FUNCTION_BLOCK FB_XPlanarModule
VAR CONSTANT
	MoverCount	 : UDINT := 2;
	TrackCount	 : UDINT := 2;
	StationCount : UDINT := 2;
END_VAR

VAR
	XPlanarSystem	: FB_Component_XPlanar;
	Movers			: ARRAY[1..MoverCount] OF FB_XPlanarMover;
	Tracks			: ARRAY[1..TrackCount] OF FB_XPlanarTrackSegment;
	Stations		: ARRAY[1..StationCount] OF FB_XPlanarStationBase;
	Station1Process : FB_SimulateProcess;  //Custom process FB that can be assigned to a station
	Station2Process : FB_RotateStation;
	InitState		: (CheckForXPlanarInit, UpdateDynamics, SetStationParameters, Initialized);
END_VAR

METHOD CyclicLogic : BOOL
VAR
	i : UDINT;
END_VAR
VAR_INST
	TaskResult	: I_PlanarTaskResult;
END_VAR
XPlanarSystem.CyclicLogic();
IF NOT XPlanarSystem.Initialized THEN
	RETURN;
END_IF

//Add any logic that needs to be called every cycle here
END_METHOD

METHOD Disable : BOOL
VAR_INST
	CommandResult	: I_PlanarTaskResult;
END_VAR
CommandResult := XPlanarSystem.Abort(); // Stop Motion and Disable All Movers
IF CommandResult.Done THEN
	Disable := TRUE;
END_IF
END_METHOD

METHOD Execute : BOOL
VAR
	i : UDINT;
END_VAR
//System is 'running' cycle thru all of the stations
FOR i := 1 TO XPlanar.StationCount DO
	ip.Stations[i].Execute();
END_FOR
END_METHOD

METHOD Initialize : BOOL
VAR_INST
	i			: UDINT;
END_VAR
CASE InitState OF
	CheckForXPlanarInit: // Init Vars
		Initialize := FALSE;
		
		//Make sure the XPlanar motion system has initialized
		IF XPlanarSystem.Initialized THEN
			InitState := UpdateDynamics;
		END_IF

	UpdateDynamics: 
		//Assign Initial Application Mover Dynamics
		FOR i := 1 TO XPlanar.MoverCount DO
			ip.Movers[i].Gap						:= 200;
			ip.Movers[i].Dynamics.Movement.Velocity := GVL.MoverVelo;
			ip.Movers[i].Dynamics.Movement.Accel	:= GVL.MoverVelo * 10;
			ip.Movers[i].Dynamics.Movement.Decel	:= GVL.MoverVelo * 10;
			ip.Movers[i].Dynamics.Movement.Jerk		:= GVL.MoverVelo * 100;
			ip.Movers[i].Dynamics.Rotation.Velocity := GVL.MoverSpinVelo;
			ip.Movers[i].Dynamics.Rotation.Accel	:= GVL.MoverSpinVelo * 10;
			ip.Movers[i].Dynamics.Rotation.Decel	:= GVL.MoverSpinVelo * 10;
			ip.Movers[i].Dynamics.Rotation.Jerk		:= GVL.MoverSpinVelo * 100;
		END_FOR

		InitState := SetStationParameters;

	SetStationParameters:
		IF SetupStations() THEN
			InitState := Initialized;
		END_IF

	Initialized: // Init Complete
		Initialize := TRUE;
END_CASE
END_METHOD

METHOD Recovery : BOOL
VAR_INST
	nState			: UDINT;
	ipResult		: ARRAY[1..MoverCount] OF I_PlanarTaskResult;
	ErrorMoverId, i : UDINT;
	ItemsOk			: BOOL;
END_VAR
//This is an example of some very simple mover recovery.  
//What needs to be done to recover will be unique for each application.

CASE nState OF
	0: // Init Vars
		Recovery := FALSE;
		i := 1;
		NextStep(nState);
		
	10: // All Movers Join rack closest to their current location
		IF i <= XPlanar.MoverCount THEN
			ipResult[i] := ip.Movers[i].MoveCommand.JoinClosestTrack(FALSE);
			IF ipResult[i].Done THEN
				NextMinorStep(nState);
			ELSIF ipResult[i].Error THEN
				ErrorStep(nState);
			END_IF
		ELSE
			i := 1;
			NextStep(nState);
		END_IF

	11: //Check Mover Count
		IF i <= XPlanar.MoverCount THEN
			i	   := i + 1;
			nState := 10;
		ELSE
			i := 1;
			NextStep(nState);
		END_IF

	20: // Sort and send Movers to Stations
		FOR i := 1 TO XPlanar.MoverCount DO
			ipResult[i] := ip.Movers[i].MoveCommand.SendToStation(ip.Stations[1]);
		END_FOR

		NextStep(nState);

	30: // Wait For Mover to Move
		ItemsOk := TRUE;
		FOR i := 1 TO XPlanar.MoverCount DO
			IF NOT ipResult[i].Busy THEN
				ItemsOk := FALSE;
			END_IF

			IF ipResult[i].Error THEN
				ErrorMoverId := i;
				ErrorStep(nState);
			END_IF
		END_FOR

		IF ItemsOk THEN
			ErrorMoverId := 0;
			NextStep(nState);
		END_IF

	40: // Complete
		nState		 := 0;
		ErrorMoverId := 0;
		Recovery	 := TRUE;
END_CASE
END_METHOD

METHOD Reset : BOOL
VAR_INST
	nState		  : UDINT;
	i			  : UDINT;
	ResetOk		  : BOOL;
	ResetError	  : BOOL;
	CommandResult : I_PlanarTaskResult;
END_VAR
CASE nState OF
	0: // Init Vars
		Reset := FALSE;
		NextStep(nState);

	10: // Reset Table 
		IF XPlanarSystem.Reset().Done THEN
			NextStep(nState);
		END_IF

	20: // Reset Stations
		FOR i := 1 TO StationCount DO
			ip.Stations[i].Reset();
		END_FOR

		NextStep(nState);

	30: // Enable Movers
		CommandResult := XPlanarSystem.EnableMovers();
		IF CommandResult.Done THEN
			NextStep(nState);
		ELSIF CommandResult.Error THEN
			ErrorStep(nState);
		END_IF

	40: // Add Movers To Group
		CommandResult := XPlanarSystem.AddMoversToGroup();
		IF CommandResult.Done THEN
			NextStep(nState);
		ELSIF CommandResult.Error THEN
			ErrorStep(nState);
		END_IF

	50: // Enable Tracks
		CommandResult := XPlanarSystem.EnableTracks();
		IF CommandResult.Done THEN
			NextStep(nState);
		ELSIF CommandResult.Error THEN
			ErrorStep(nState);
		END_IF

	60: // Add Tracks To Group
		CommandResult := XPlanarSystem.AddTracksToGroup();
		IF CommandResult.Done THEN
			NextStep(nState);
		ELSIF CommandResult.Error THEN
			ErrorStep(nState);
		END_IF

	70: // Enable Group
		CommandResult := XPlanarSystem.EnableGroup();
		IF CommandResult.Done THEN
			NextStep(nState);
		ELSIF CommandResult.Error THEN
			ErrorStep(nState);
		END_IF

	80: // Complete
		Reset  := TRUE;
		nState := 0;
END_CASE
END_METHOD

METHOD PRIVATE SetupStations : BOOL
// Setup Station 1
Stations[1].ID := 1;
Stations[1].TrackID := 1;
Stations[1].Position.SetValuesXYC(120, 60, 0);
Stations[1].NextStation := ip.Stations[2];
Stations[1].Process := Station1Process; //Assign a custom process to the station
Station1Process.ProcessTime := 1.5;


// Setup Station 2
Stations[2].ID := 2;
Stations[2].TrackID := 2;
Stations[2].Position.SetValuesXYC(120, 360, 0);
Stations[2].NextStation := ip.Stations[1];
Stations[2].Process := Station2Process; //Assign a custom process to the station
Station2Process.NumberOfTurns := 2;
Station2Process.StationAngle := 0;


SetupStations:=TRUE;
END_METHOD

END_FUNCTION_BLOCK

(* stored: Version 1.1.0.1
   POU FB_XPlanarModule: Id {fc8a5627-8159-4948-be60-7bb109013f17}, SpecialFunc None
   Method CyclicLogic: Id {29a5b2a6-b906-481e-b2a5-9e6b8b00dcb1}
   Method Disable: Id {bea64788-04c2-46d8-901f-da40359402f9}
   Method Execute: Id {e9c18260-d963-4b3b-9ac1-c7c999f6e501}
   Method Initialize: Id {68346b41-b68e-48f0-9612-b8cb0e4f6801}
   Method Recovery: Id {a9841bea-60cb-426f-bc44-b8cede3e8fbc}
   Method Reset: Id {77b1ac13-4d41-4ec9-b757-dd7d7db44fa5}
   Method SetupStations: Id {15ffb126-4413-4503-9c58-ae49f83f5dbf} *)
